{attribute 'linkalways'} 
{attribute 'no_explicit_call' := 'This FB is a CLASS and must be accessed using methods or properties'}
{attribute 'enable_dynamic_creation'}
FUNCTION_BLOCK PUBLIC DeserializationFailedNodeNotSupportedAlarm EXTENDS Alarm
VAR
	state : (CLEARED, RAISED);
	_reason : T_MAXSTRING;
END_VAR

PROPERTY Active : BOOL
GET
Active := state <> CLEARED;
END_GET
END_PROPERTY

METHOD PUBLIC Clear
_reason := '';
state := CLEARED;
END_METHOD

PROPERTY PUBLIC Message : T_MaxString
GET
Message := 'Node type is not installed';
END_GET
END_PROPERTY

METHOD PUBLIC Raise
VAR_INPUT
	NodeType : T_MAXSTRING;
END_VAR
_reason := NodeType;
state := RAISED;
END_METHOD

PROPERTY Reason : T_MaxString
GET
Reason := _reason;
END_GET
END_PROPERTY

END_FUNCTION_BLOCK

(* stored: Version 1.1.0.1, ProductVersion 3.1.4024.12
   POU DeserializationFailedNodeNotSupportedAlarm: Id {9623ea07-68e6-068a-1ae8-7c1b189690f8}, SpecialFunc None
   Property Active: Id {662c13d9-0379-0ff6-0cc0-325aad0e11ed}
   Get Get: Id {16e3e2a6-2852-0e19-1d26-92eb36f05ea1}
   Method Clear: Id {63f4bc84-c70c-0daa-2e5a-8f3ae0175326}
   Property Message: Id {a8f7f573-e6f1-0ec2-0054-980ab27da1ae}
   Get Get: Id {b61a98d1-a834-06e5-18b6-698db9d9e9ba}
   Method Raise: Id {85c61a4a-d853-09be-378f-20a8832e1ec7}
   Property Reason: Id {44b8d335-4271-063a-2ae7-6ff7902b06a9}
   Get Get: Id {85e5fb5f-cdb9-058f-3ca8-1f45cd93f658} *)
